// TIA Portal V20 export
TYPE "TypeHeaderPlc"
   STRUCT
      conActive : Bool;   // connection is established
      err : Bool;   // fault general
      errWd : Bool;   // fault watchdog
      errSd : Bool;   // fault send
      errRd : Bool;   // fault receive
      bit05 : Bool;
      bit06 : Bool;
      bit07 : Bool;
      sdBusy : Bool;   // new data is sending
      sdDone : Bool;   // new data sended
      rdBusy : Bool;   // new data is receiving
      rdDone : Bool;   // new data received
      sdOverload : Bool;   // new data could not be sent because the Cp overloaded
      statistic : Bool;   // statistic information are aviable
      bit16 : Bool;
      bit17 : Bool;
      sdState : Word;   // send state
      sdLastErrState : Word;   // send last fault state
      sdLenght : Int;   // send lenght [byte]
      sdCps : Int;   // send counter per second
      rdState : Word;   // receive state
      rdLastErrState : Word;   // receive last fault state
      rdLenght : Int;   // receive lenght [byte]
      rdCps : Int;   // receive counter per second
      in18 : Int;
   END_STRUCT;
END_TYPE
